% RSLogix 500 project LCDTEST_BAK006.RSS, saved by version 8.10.00.30 %
PROJECT "UNTITLED"    % processor: Bul.1763 MicroLogix 1100 Series B %

PROGRAM FILES
  LAD 2   3 rungs

DATA FILES
  O0 OUTPUT  4 elements
  I1 INPUT  6 elements
  S2 STATUS  66 elements
  B3 BINARY  1 elements
  T4 TIMER  1 elements
  C5 COUNTER  1 elements
  R6 CONTROL  1 elements
  N7 INTEGER  1 elements
  F8 FLOAT  1 elements
  ST9 ST9  6 elements

LADDER 2
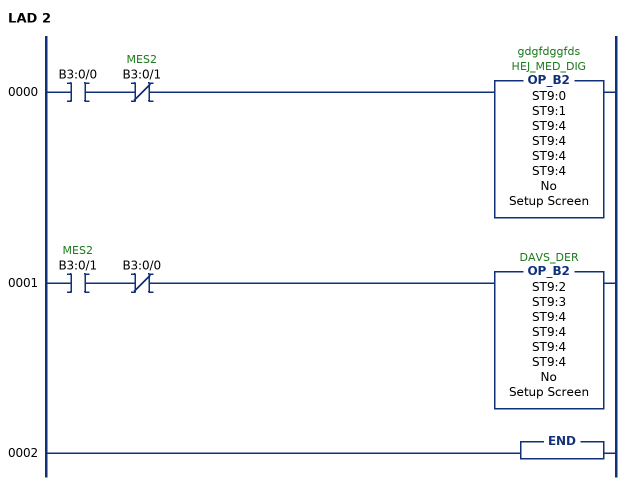
% Rung: 0 %
SOR XIC B3:0/0 XIO B3:0/1 OP_B2 ST9:0 ST9:1 ST9:4 ST9:4 ST9:4 ST9:4 No "Setup Screen" EOR
%   B3:0/1  MES2 %
%   ST9:0  HEJ_MED_DIG  "gdgfdggfds" %
%   ST9:1  HOW_R_U %
% Rung: 1 %
SOR XIC B3:0/1 XIO B3:0/0 OP_B2 ST9:2 ST9:3 ST9:4 ST9:4 ST9:4 ST9:4 No "Setup Screen" EOR
%   B3:0/1  MES2 %
%   ST9:2  DAVS_DER %
% Rung: 2 %
SOR END EOR

OTHER DOCUMENTED ADDRESSES
  B3:0  MES1

DATA TABLE (non-zero values as saved)
DATA B3
% B3:0 % 0X0002
